(* IEC 61131-3 sources: RL_MAR/experiments/comparison/autoplc/results/qwen3.5-9b_20260511_180311/med_35, 1 file *)

(* ---- med_35_1.st ---- *)
FUNCTION_BLOCK FB_SimpleCalculation
VAR_INPUT
INPUT_VAR1 : INT := 2;
VAR2 : INT := 0;
END_VAR

VAR_OUTPUT
OUTPUT_VAR1 : INT;
OUTPUT_VAR2 : INT;
END_VAR

VAR
COUNTER2 : INT := 0;
TEMP_VAR1 : INT;
TEMP_VAR2 : INT;
I : INT;
END_VAR

END_FUNCTION_BLOCK
